// Mitsubishi GX Developer project: 中間搬送   PLC: Q02

PROGRAM MAIN
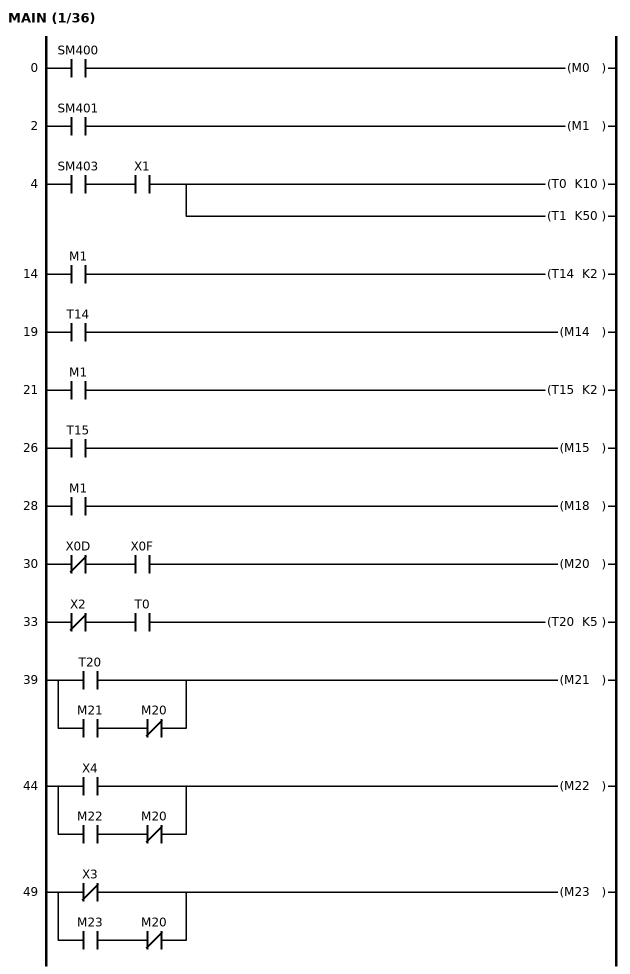
0     LD      SM400
      OUT     M0
2     LD      SM401
      OUT     M1
4     LD      SM403
      AND     X1
      OUT     T0 K10
      OUT     T1 K50
14    LD      M1
      OUT     T14 K2
19    LD      T14
      OUT     M14
21    LD      M1
      OUT     T15 K2
26    LD      T15
      OUT     M15
28    LD      M1
      OUT     M18
30    LDI     X0D
      AND     X0F
      OUT     M20
33    LDI     X2
      AND     T0
      OUT     T20 K5
39    LD      T20
      LD      M21
      ANI     M20
      ORB
      OUT     M21
44    LD      X4
      LD      M22
      ANI     M20
      ORB
      OUT     M22
49    LDI     X3
      LD      M23
      ANI     M20
      ORB
      OUT     M23
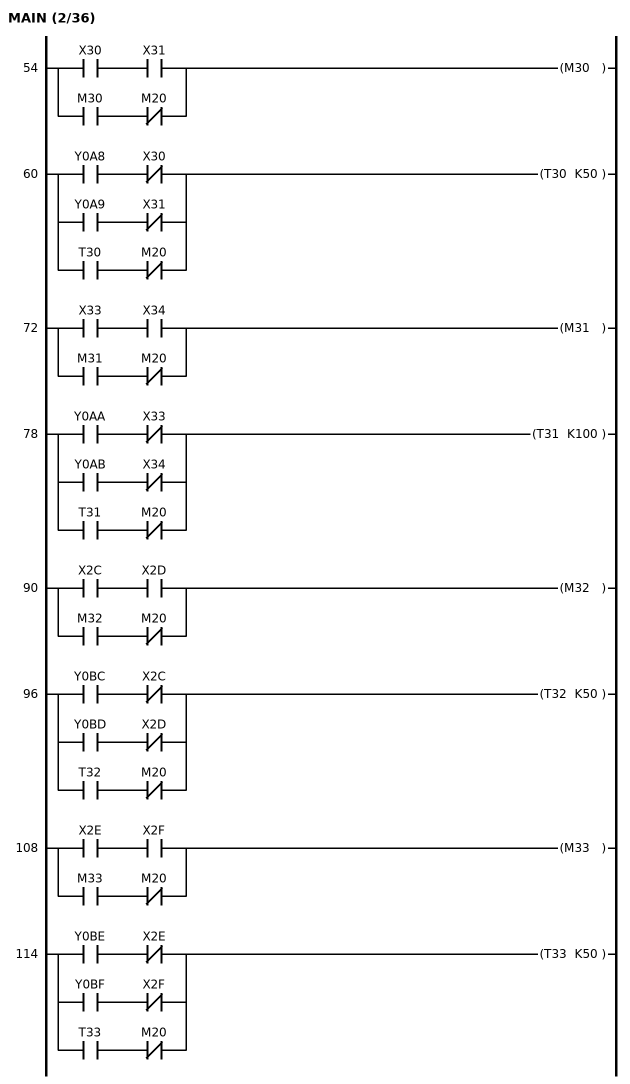
54    LD      X30
      AND     X31
      LD      M30
      ANI     M20
      ORB
      OUT     M30
60    LD      Y0A8
      ANI     X30
      LD      Y0A9
      ANI     X31
      ORB
      LD      T30
      ANI     M20
      ORB
      OUT     T30 K50
72    LD      X33
      AND     X34
      LD      M31
      ANI     M20
      ORB
      OUT     M31
78    LD      Y0AA
      ANI     X33
      LD      Y0AB
      ANI     X34
      ORB
      LD      T31
      ANI     M20
      ORB
      OUT     T31 K100
90    LD      X2C
      AND     X2D
      LD      M32
      ANI     M20
      ORB
      OUT     M32
96    LD      Y0BC
      ANI     X2C
      LD      Y0BD
      ANI     X2D
      ORB
      LD      T32
      ANI     M20
      ORB
      OUT     T32 K50
108   LD      X2E
      AND     X2F
      LD      M33
      ANI     M20
      ORB
      OUT     M33
114   LD      Y0BE
      ANI     X2E
      LD      Y0BF
      ANI     X2F
      ORB
      LD      T33
      ANI     M20
      ORB
      OUT     T33 K50
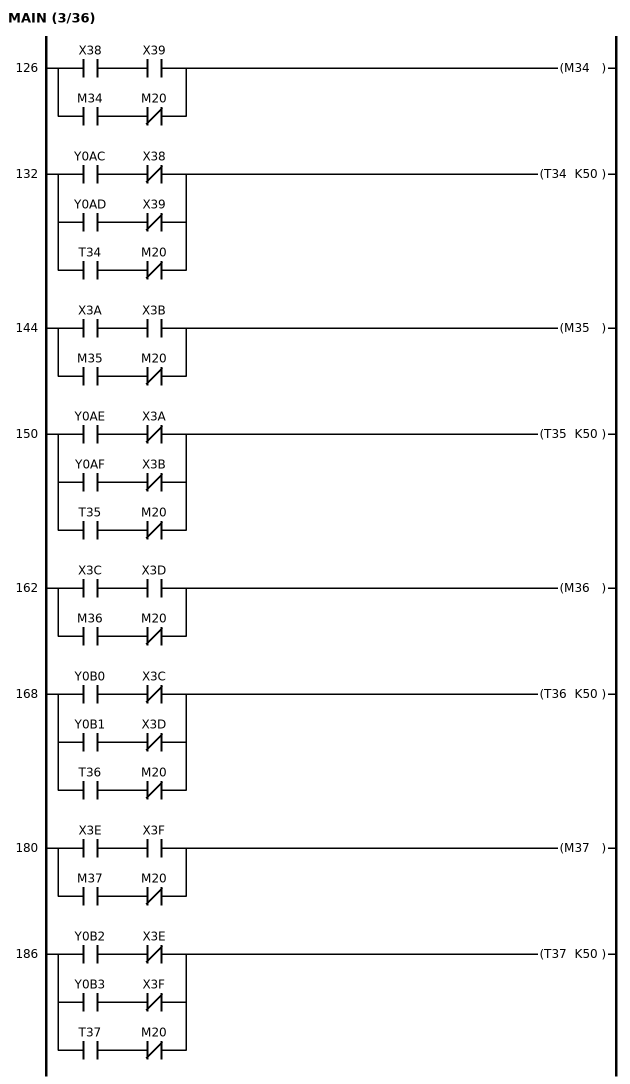
126   LD      X38
      AND     X39
      LD      M34
      ANI     M20
      ORB
      OUT     M34
132   LD      Y0AC
      ANI     X38
      LD      Y0AD
      ANI     X39
      ORB
      LD      T34
      ANI     M20
      ORB
      OUT     T34 K50
144   LD      X3A
      AND     X3B
      LD      M35
      ANI     M20
      ORB
      OUT     M35
150   LD      Y0AE
      ANI     X3A
      LD      Y0AF
      ANI     X3B
      ORB
      LD      T35
      ANI     M20
      ORB
      OUT     T35 K50
162   LD      X3C
      AND     X3D
      LD      M36
      ANI     M20
      ORB
      OUT     M36
168   LD      Y0B0
      ANI     X3C
      LD      Y0B1
      ANI     X3D
      ORB
      LD      T36
      ANI     M20
      ORB
      OUT     T36 K50
180   LD      X3E
      AND     X3F
      LD      M37
      ANI     M20
      ORB
      OUT     M37
186   LD      Y0B2
      ANI     X3E
      LD      Y0B3
      ANI     X3F
      ORB
      LD      T37
      ANI     M20
      ORB
      OUT     T37 K50
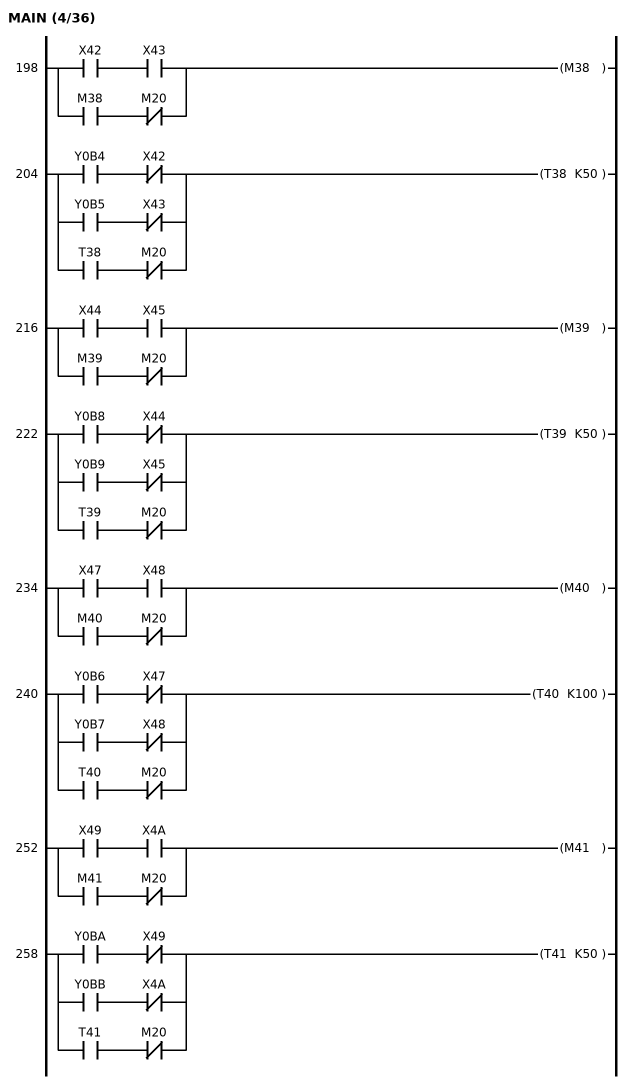
198   LD      X42
      AND     X43
      LD      M38
      ANI     M20
      ORB
      OUT     M38
204   LD      Y0B4
      ANI     X42
      LD      Y0B5
      ANI     X43
      ORB
      LD      T38
      ANI     M20
      ORB
      OUT     T38 K50
216   LD      X44
      AND     X45
      LD      M39
      ANI     M20
      ORB
      OUT     M39
222   LD      Y0B8
      ANI     X44
      LD      Y0B9
      ANI     X45
      ORB
      LD      T39
      ANI     M20
      ORB
      OUT     T39 K50
234   LD      X47
      AND     X48
      LD      M40
      ANI     M20
      ORB
      OUT     M40
240   LD      Y0B6
      ANI     X47
      LD      Y0B7
      ANI     X48
      ORB
      LD      T40
      ANI     M20
      ORB
      OUT     T40 K100
252   LD      X49
      AND     X4A
      LD      M41
      ANI     M20
      ORB
      OUT     M41
258   LD      Y0BA
      ANI     X49
      LD      Y0BB
      ANI     X4A
      ORB
      LD      T41
      ANI     M20
      ORB
      OUT     T41 K50
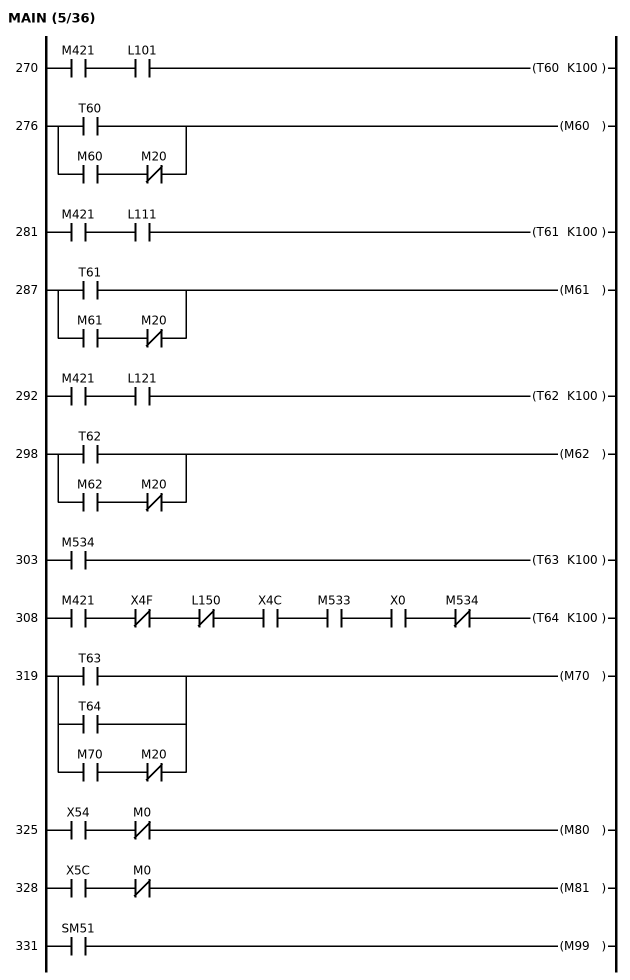
270   LD      M421
      AND     L101
      OUT     T60 K100
276   LD      T60
      LD      M60
      ANI     M20
      ORB
      OUT     M60
281   LD      M421
      AND     L111
      OUT     T61 K100
287   LD      T61
      LD      M61
      ANI     M20
      ORB
      OUT     M61
292   LD      M421
      AND     L121
      OUT     T62 K100
298   LD      T62
      LD      M62
      ANI     M20
      ORB
      OUT     M62
303   LD      M534
      OUT     T63 K100
308   LD      M421
      ANI     X4F
      ANI     L150
      AND     X4C
      AND     M533
      AND     X0
      ANI     M534
      OUT     T64 K100
319   LD      T63
      OR      T64
      LD      M70
      ANI     M20
      ORB
      OUT     M70
325   LD      X54
      ANI     M0
      OUT     M80
328   LD      X5C
      ANI     M0
      OUT     M81
331   LD      SM51
      OUT     M99
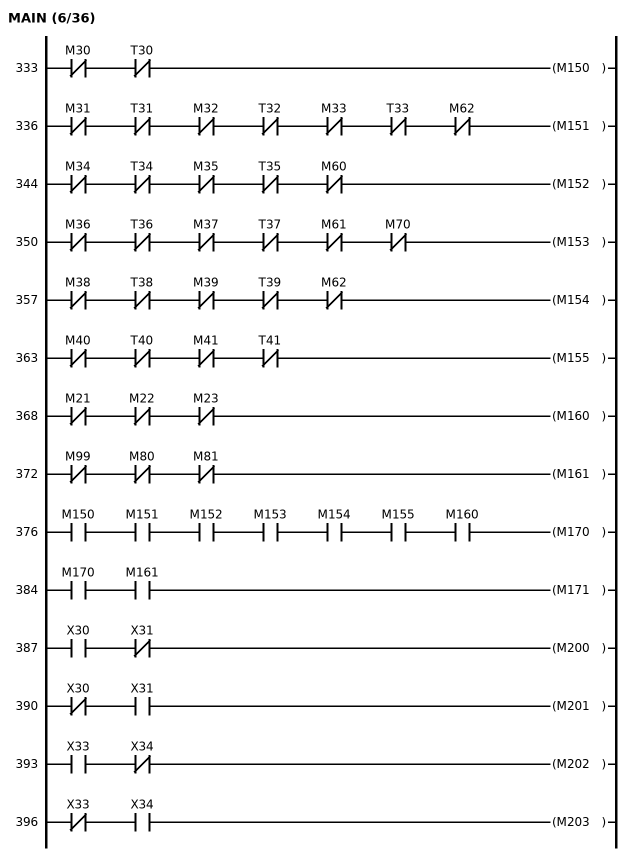
333   LDI     M30
      ANI     T30
      OUT     M150
336   LDI     M31
      ANI     T31
      ANI     M32
      ANI     T32
      ANI     M33
      ANI     T33
      ANI     M62
      OUT     M151
344   LDI     M34
      ANI     T34
      ANI     M35
      ANI     T35
      ANI     M60
      OUT     M152
350   LDI     M36
      ANI     T36
      ANI     M37
      ANI     T37
      ANI     M61
      ANI     M70
      OUT     M153
357   LDI     M38
      ANI     T38
      ANI     M39
      ANI     T39
      ANI     M62
      OUT     M154
363   LDI     M40
      ANI     T40
      ANI     M41
      ANI     T41
      OUT     M155
368   LDI     M21
      ANI     M22
      ANI     M23
      OUT     M160
372   LDI     M99
      ANI     M80
      ANI     M81
      OUT     M161
376   LD      M150
      AND     M151
      AND     M152
      AND     M153
      AND     M154
      AND     M155
      AND     M160
      OUT     M170
384   LD      M170
      AND     M161
      OUT     M171
387   LD      X30
      ANI     X31
      OUT     M200
390   LDI     X30
      AND     X31
      OUT     M201
393   LD      X33
      ANI     X34
      OUT     M202
396   LDI     X33
      AND     X34
      OUT     M203
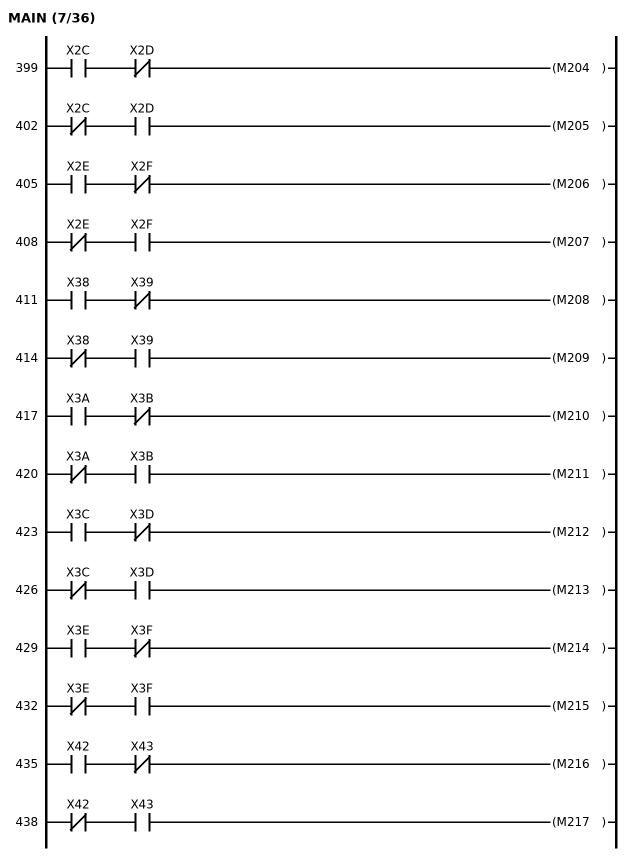
399   LD      X2C
      ANI     X2D
      OUT     M204
402   LDI     X2C
      AND     X2D
      OUT     M205
405   LD      X2E
      ANI     X2F
      OUT     M206
408   LDI     X2E
      AND     X2F
      OUT     M207
411   LD      X38
      ANI     X39
      OUT     M208
414   LDI     X38
      AND     X39
      OUT     M209
417   LD      X3A
      ANI     X3B
      OUT     M210
420   LDI     X3A
      AND     X3B
      OUT     M211
423   LD      X3C
      ANI     X3D
      OUT     M212
426   LDI     X3C
      AND     X3D
      OUT     M213
429   LD      X3E
      ANI     X3F
      OUT     M214
432   LDI     X3E
      AND     X3F
      OUT     M215
435   LD      X42
      ANI     X43
      OUT     M216
438   LDI     X42
      AND     X43
      OUT     M217
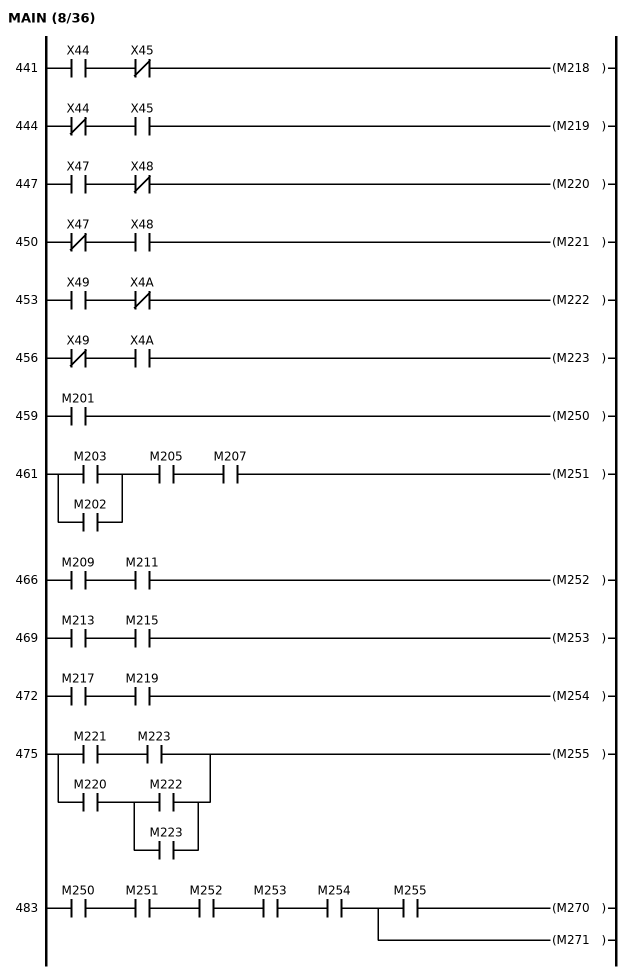
441   LD      X44
      ANI     X45
      OUT     M218
444   LDI     X44
      AND     X45
      OUT     M219
447   LD      X47
      ANI     X48
      OUT     M220
450   LDI     X47
      AND     X48
      OUT     M221
453   LD      X49
      ANI     X4A
      OUT     M222
456   LDI     X49
      AND     X4A
      OUT     M223
459   LD      M201
      OUT     M250
461   LD      M203
      OR      M202
      AND     M205
      AND     M207
      OUT     M251
466   LD      M209
      AND     M211
      OUT     M252
469   LD      M213
      AND     M215
      OUT     M253
472   LD      M217
      AND     M219
      OUT     M254
475   LD      M221
      AND     M223
      LD      M220
      LD      M222
      OR      M223
      ANB
      ORB
      OUT     M255
483   LD      M250
      AND     M251
      AND     M252
      AND     M253
      AND     M254
      MPS
      AND     M255
      OUT     M270
      MPP
      OUT     M271
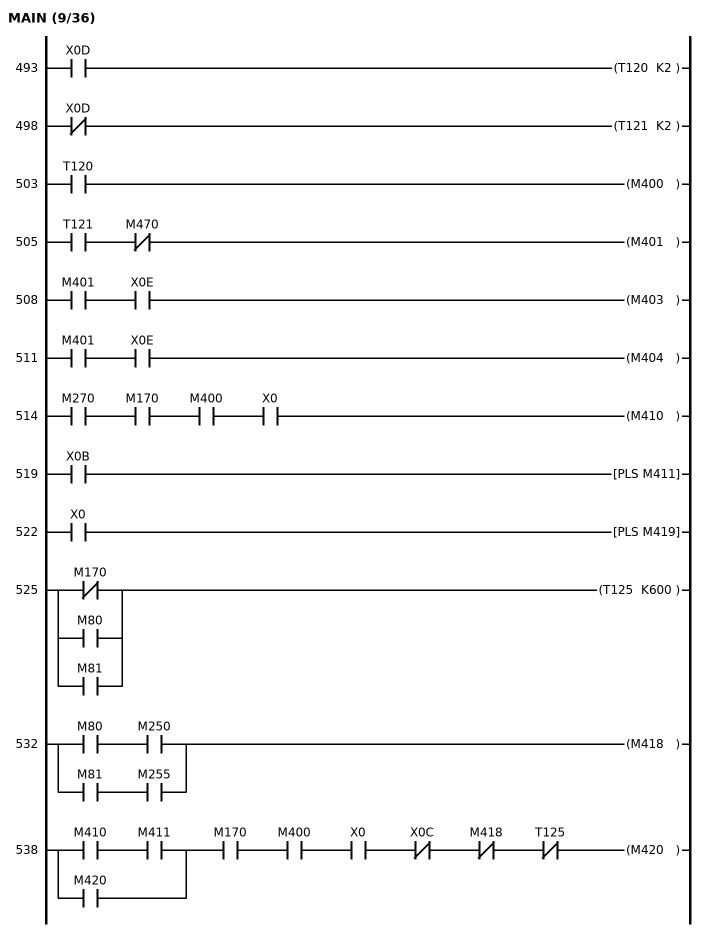
493   LD      X0D
      OUT     T120 K2
498   LDI     X0D
      OUT     T121 K2
503   LD      T120
      OUT     M400
505   LD      T121
      ANI     M470
      OUT     M401
508   LD      M401
      AND     X0E
      OUT     M403
511   LD      M401
      AND     X0E
      OUT     M404
514   LD      M270
      AND     M170
      AND     M400
      AND     X0
      OUT     M410
519   LD      X0B
      PLS     M411
522   LD      X0
      PLS     M419
525   LDI     M170
      OR      M80
      OR      M81
      OUT     T125 K600
532   LD      M80
      AND     M250
      LD      M81
      AND     M255
      ORB
      OUT     M418
538   LD      M410
      AND     M411
      OR      M420
      AND     M170
      AND     M400
      AND     X0
      ANI     X0C
      ANI     M418
      ANI     T125
      OUT     M420
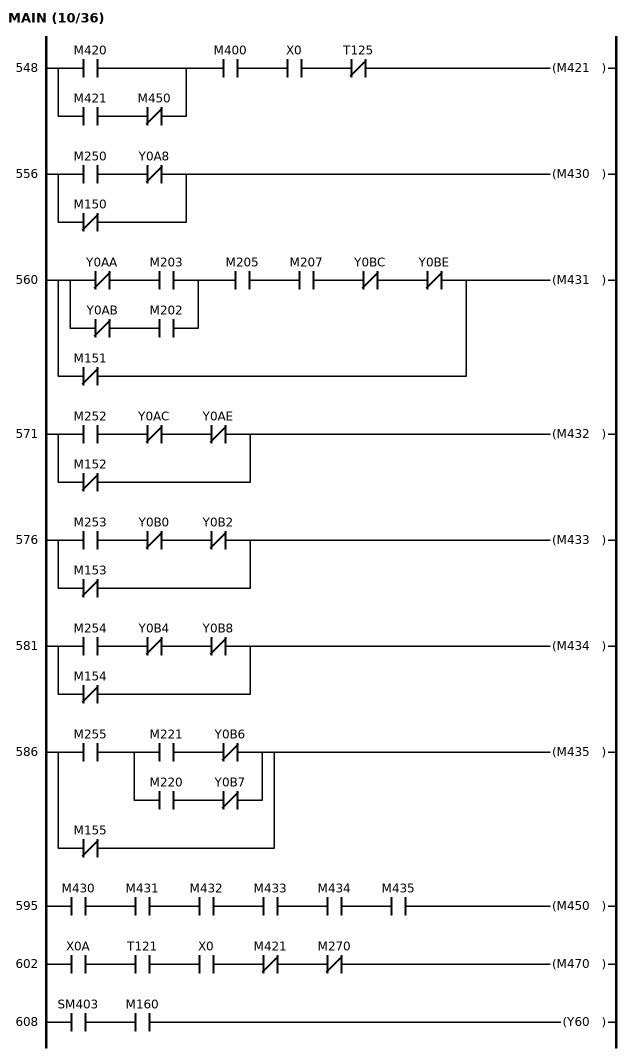
548   LD      M420
      LD      M421
      ANI     M450
      ORB
      AND     M400
      AND     X0
      ANI     T125
      OUT     M421
556   LD      M250
      ANI     Y0A8
      ORI     M150
      OUT     M430
560   LDI     Y0AA
      AND     M203
      LDI     Y0AB
      AND     M202
      ORB
      AND     M205
      AND     M207
      ANI     Y0BC
      ANI     Y0BE
      ORI     M151
      OUT     M431
571   LD      M252
      ANI     Y0AC
      ANI     Y0AE
      ORI     M152
      OUT     M432
576   LD      M253
      ANI     Y0B0
      ANI     Y0B2
      ORI     M153
      OUT     M433
581   LD      M254
      ANI     Y0B4
      ANI     Y0B8
      ORI     M154
      OUT     M434
586   LD      M255
      LD      M221
      ANI     Y0B6
      LD      M220
      ANI     Y0B7
      ORB
      ANB
      ORI     M155
      OUT     M435
595   LD      M430
      AND     M431
      AND     M432
      AND     M433
      AND     M434
      AND     M435
      OUT     M450
602   LD      X0A
      AND     T121
      AND     X0
      ANI     M421
      ANI     M270
      OUT     M470
608   LD      SM403
      AND     M160
      OUT     Y60
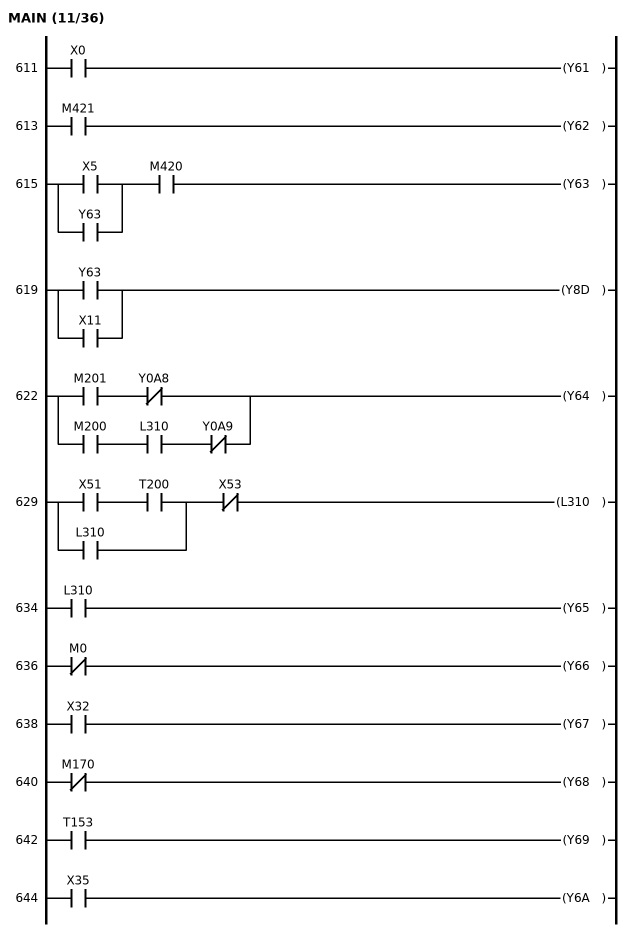
611   LD      X0
      OUT     Y61
613   LD      M421
      OUT     Y62
615   LD      X5
      OR      Y63
      AND     M420
      OUT     Y63
619   LD      Y63
      OR      X11
      OUT     Y8D
622   LD      M201
      ANI     Y0A8
      LD      M200
      AND     L310
      ANI     Y0A9
      ORB
      OUT     Y64
629   LD      X51
      AND     T200
      OR      L310
      ANI     X53
      OUT     L310
634   LD      L310
      OUT     Y65
636   LDI     M0
      OUT     Y66
638   LD      X32
      OUT     Y67
640   LDI     M170
      OUT     Y68
642   LD      T153
      OUT     Y69
644   LD      X35
      OUT     Y6A
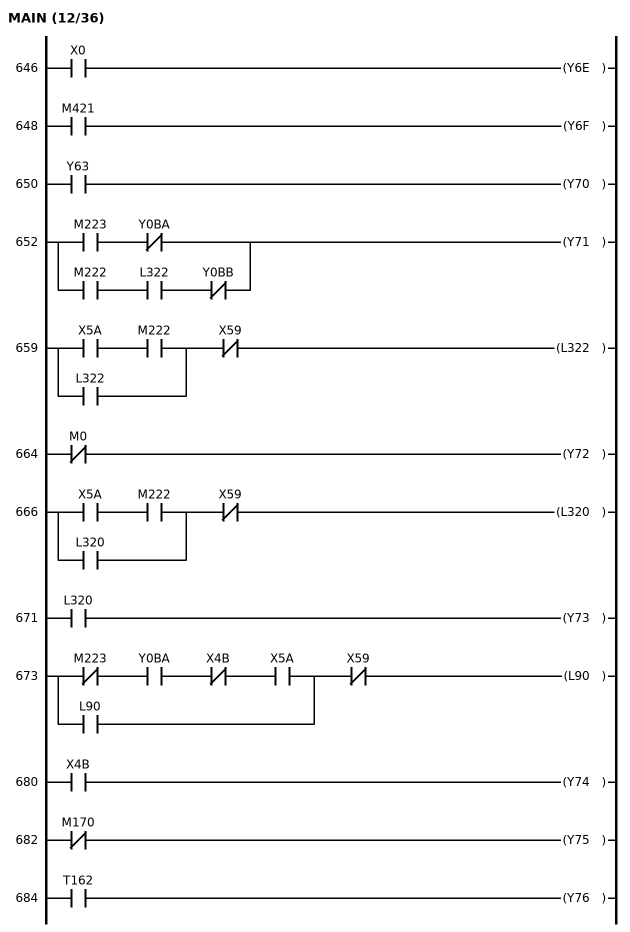
646   LD      X0
      OUT     Y6E
648   LD      M421
      OUT     Y6F
650   LD      Y63
      OUT     Y70
652   LD      M223
      ANI     Y0BA
      LD      M222
      AND     L322
      ANI     Y0BB
      ORB
      OUT     Y71
659   LD      X5A
      AND     M222
      OR      L322
      ANI     X59
      OUT     L322
664   LDI     M0
      OUT     Y72
666   LD      X5A
      AND     M222
      OR      L320
      ANI     X59
      OUT     L320
671   LD      L320
      OUT     Y73
673   LDI     M223
      AND     Y0BA
      ANI     X4B
      AND     X5A
      OR      L90
      ANI     X59
      OUT     L90
680   LD      X4B
      OUT     Y74
682   LDI     M170
      OUT     Y75
684   LD      T162
      OUT     Y76
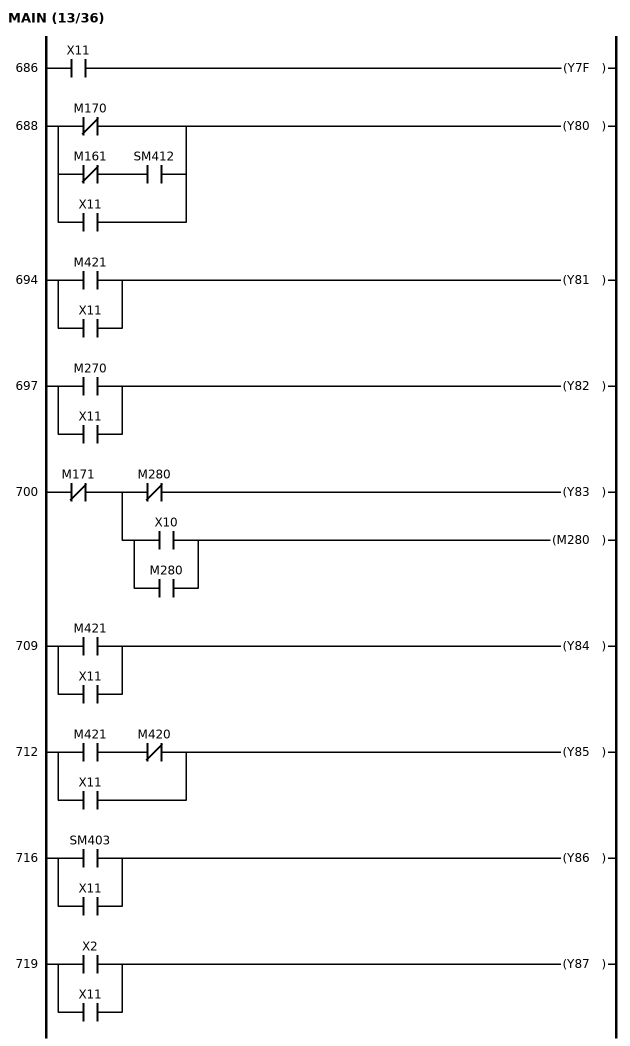
686   LD      X11
      OUT     Y7F
688   LDI     M170
      LDI     M161
      AND     SM412
      ORB
      OR      X11
      OUT     Y80
694   LD      M421
      OR      X11
      OUT     Y81
697   LD      M270
      OR      X11
      OUT     Y82
700   LDI     M171
      MPS
      ANI     M280
      OUT     Y83
      MPP
      LD      X10
      OR      M280
      ANB
      OUT     M280
709   LD      M421
      OR      X11
      OUT     Y84
712   LD      M421
      ANI     M420
      OR      X11
      OUT     Y85
716   LD      SM403
      OR      X11
      OUT     Y86
719   LD      X2
      OR      X11
      OUT     Y87
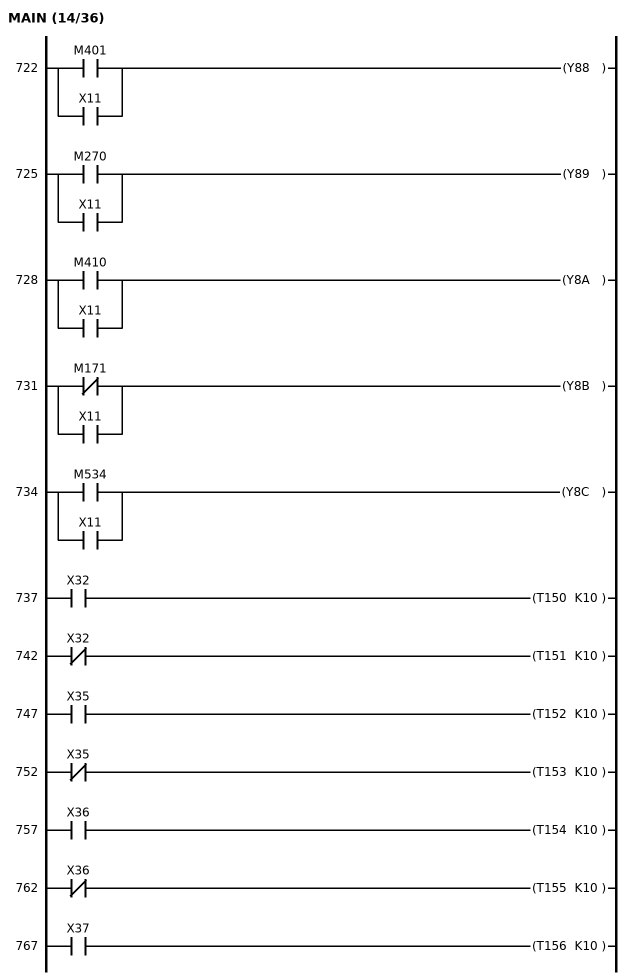
722   LD      M401
      OR      X11
      OUT     Y88
725   LD      M270
      OR      X11
      OUT     Y89
728   LD      M410
      OR      X11
      OUT     Y8A
731   LDI     M171
      OR      X11
      OUT     Y8B
734   LD      M534
      OR      X11
      OUT     Y8C
737   LD      X32
      OUT     T150 K10
742   LDI     X32
      OUT     T151 K10
747   LD      X35
      OUT     T152 K10
752   LDI     X35
      OUT     T153 K10
757   LD      X36
      OUT     T154 K10
762   LDI     X36
      OUT     T155 K10
767   LD      X37
      OUT     T156 K10
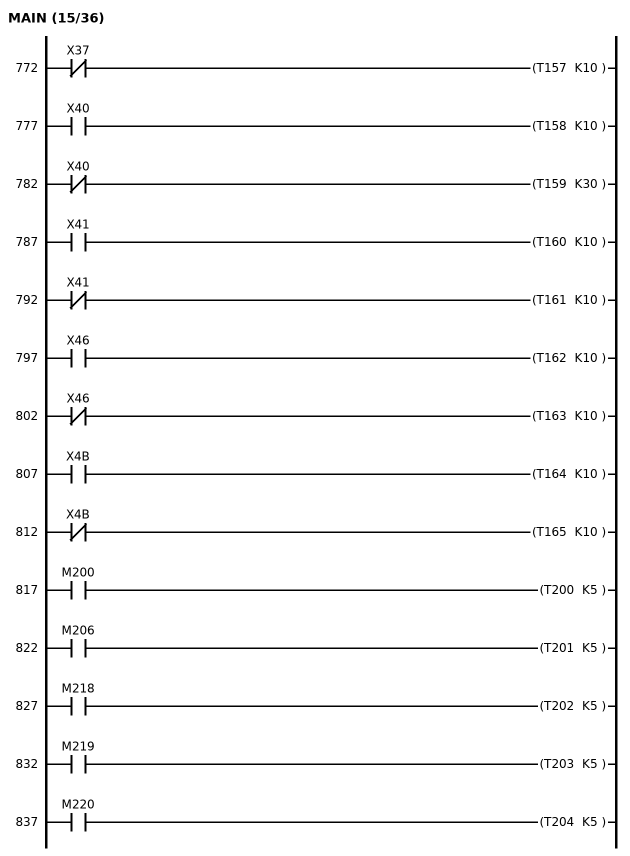
772   LDI     X37
      OUT     T157 K10
777   LD      X40
      OUT     T158 K10
782   LDI     X40
      OUT     T159 K30
787   LD      X41
      OUT     T160 K10
792   LDI     X41
      OUT     T161 K10
797   LD      X46
      OUT     T162 K10
802   LDI     X46
      OUT     T163 K10
807   LD      X4B
      OUT     T164 K10
812   LDI     X4B
      OUT     T165 K10
817   LD      M200
      OUT     T200 K5
822   LD      M206
      OUT     T201 K5
827   LD      M218
      OUT     T202 K5
832   LD      M219
      OUT     T203 K5
837   LD      M220
      OUT     T204 K5
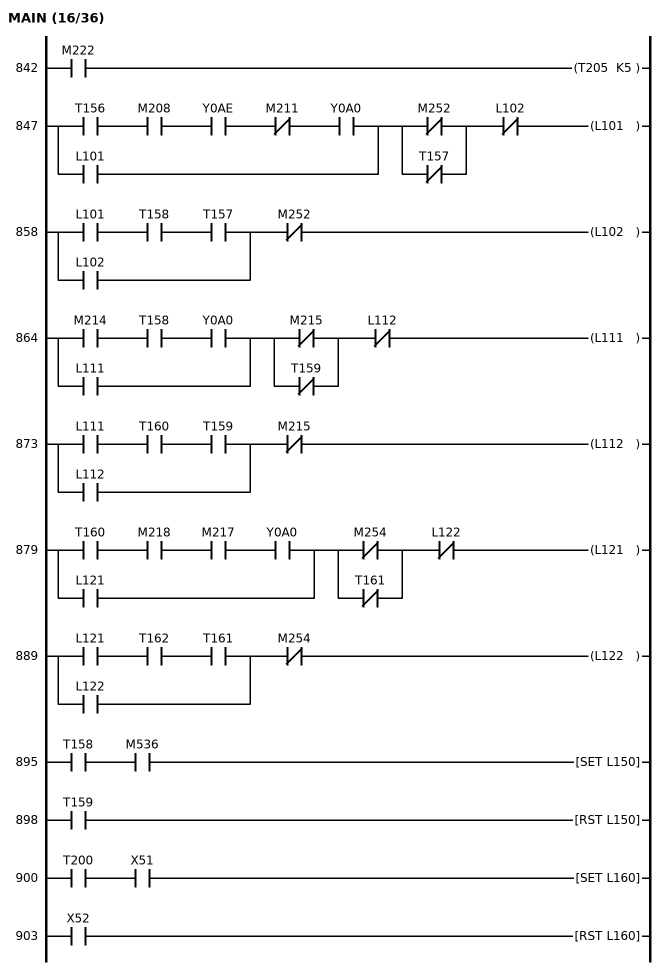
842   LD      M222
      OUT     T205 K5
847   LD      T156
      AND     M208
      AND     Y0AE
      ANI     M211
      AND     Y0A0
      OR      L101
      LDI     M252
      ORI     T157
      ANB
      ANI     L102
      OUT     L101
858   LD      L101
      AND     T158
      AND     T157
      OR      L102
      ANI     M252
      OUT     L102
864   LD      M214
      AND     T158
      AND     Y0A0
      OR      L111
      LDI     M215
      ORI     T159
      ANB
      ANI     L112
      OUT     L111
873   LD      L111
      AND     T160
      AND     T159
      OR      L112
      ANI     M215
      OUT     L112
879   LD      T160
      AND     M218
      AND     M217
      AND     Y0A0
      OR      L121
      LDI     M254
      ORI     T161
      ANB
      ANI     L122
      OUT     L121
889   LD      L121
      AND     T162
      AND     T161
      OR      L122
      ANI     M254
      OUT     L122
895   LD      T158
      AND     M536
      SET     L150
898   LD      T159
      RST     L150
900   LD      T200
      AND     X51
      SET     L160
903   LD      X52
      RST     L160
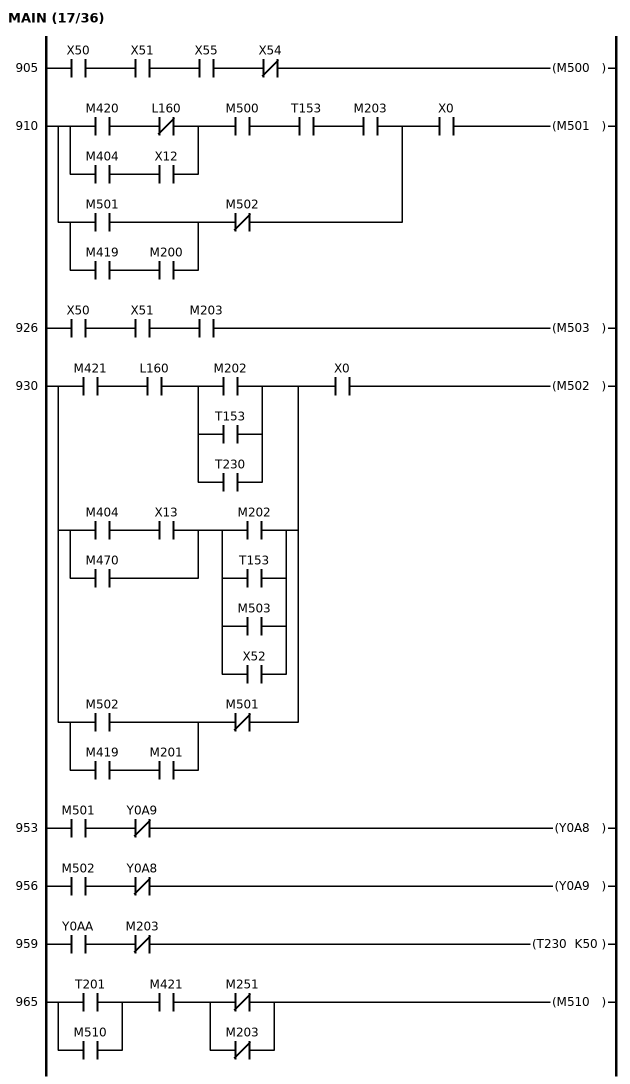
905   LD      X50
      AND     X51
      AND     X55
      ANI     X54
      OUT     M500
910   LD      M420
      ANI     L160
      LD      M404
      AND     X12
      ORB
      AND     M500
      AND     T153
      AND     M203
      LD      M501
      LD      M419
      AND     M200
      ORB
      ANI     M502
      ORB
      AND     X0
      OUT     M501
926   LD      X50
      AND     X51
      AND     M203
      OUT     M503
930   LD      M421
      AND     L160
      LD      M202
      OR      T153
      OR      T230
      ANB
      LD      M404
      AND     X13
      OR      M470
      LD      M202
      OR      T153
      OR      M503
      OR      X52
      ANB
      ORB
      LD      M502
      LD      M419
      AND     M201
      ORB
      ANI     M501
      ORB
      AND     X0
      OUT     M502
953   LD      M501
      ANI     Y0A9
      OUT     Y0A8
956   LD      M502
      ANI     Y0A8
      OUT     Y0A9
959   LD      Y0AA
      ANI     M203
      OUT     T230 K50
965   LD      T201
      OR      M510
      AND     M421
      LDI     M251
      ORI     M203
      ANB
      OUT     M510
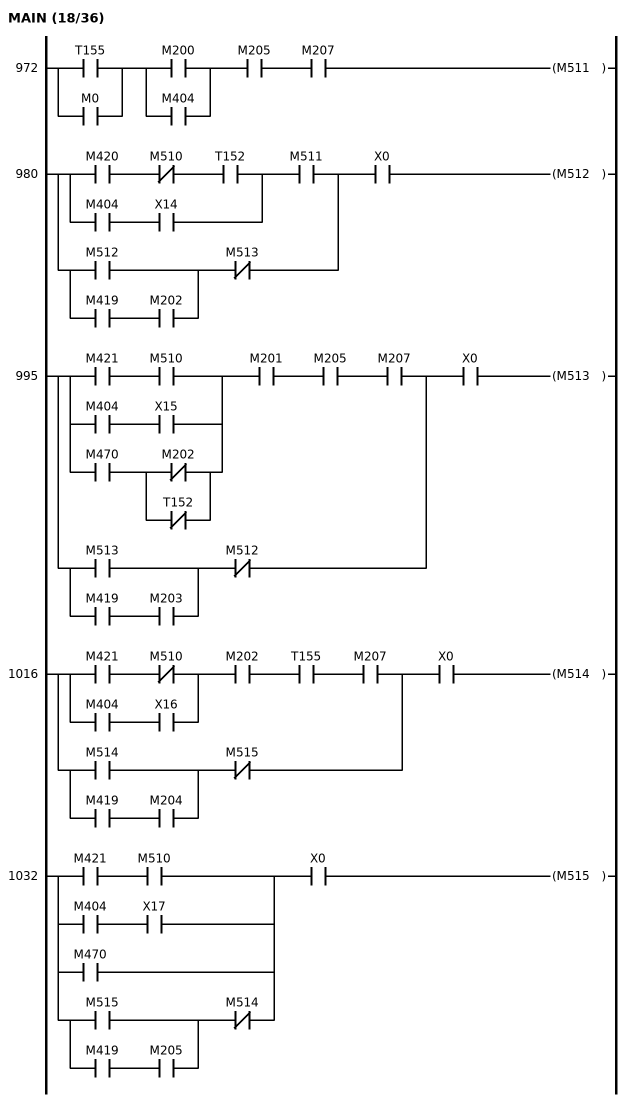
972   LD      T155
      OR      M0
      LD      M200
      OR      M404
      ANB
      AND     M205
      AND     M207
      OUT     M511
980   LD      M420
      ANI     M510
      AND     T152
      LD      M404
      AND     X14
      ORB
      AND     M511
      LD      M512
      LD      M419
      AND     M202
      ORB
      ANI     M513
      ORB
      AND     X0
      OUT     M512
995   LD      M421
      AND     M510
      LD      M404
      AND     X15
      ORB
      LD      M470
      LDI     M202
      ORI     T152
      ANB
      ORB
      AND     M201
      AND     M205
      AND     M207
      LD      M513
      LD      M419
      AND     M203
      ORB
      ANI     M512
      ORB
      AND     X0
      OUT     M513
1016  LD      M421
      ANI     M510
      LD      M404
      AND     X16
      ORB
      AND     M202
      AND     T155
      AND     M207
      LD      M514
      LD      M419
      AND     M204
      ORB
      ANI     M515
      ORB
      AND     X0
      OUT     M514
1032  LD      M421
      AND     M510
      LD      M404
      AND     X17
      ORB
      OR      M470
      LD      M515
      LD      M419
      AND     M205
      ORB
      ANI     M514
      ORB
      AND     X0
      OUT     M515
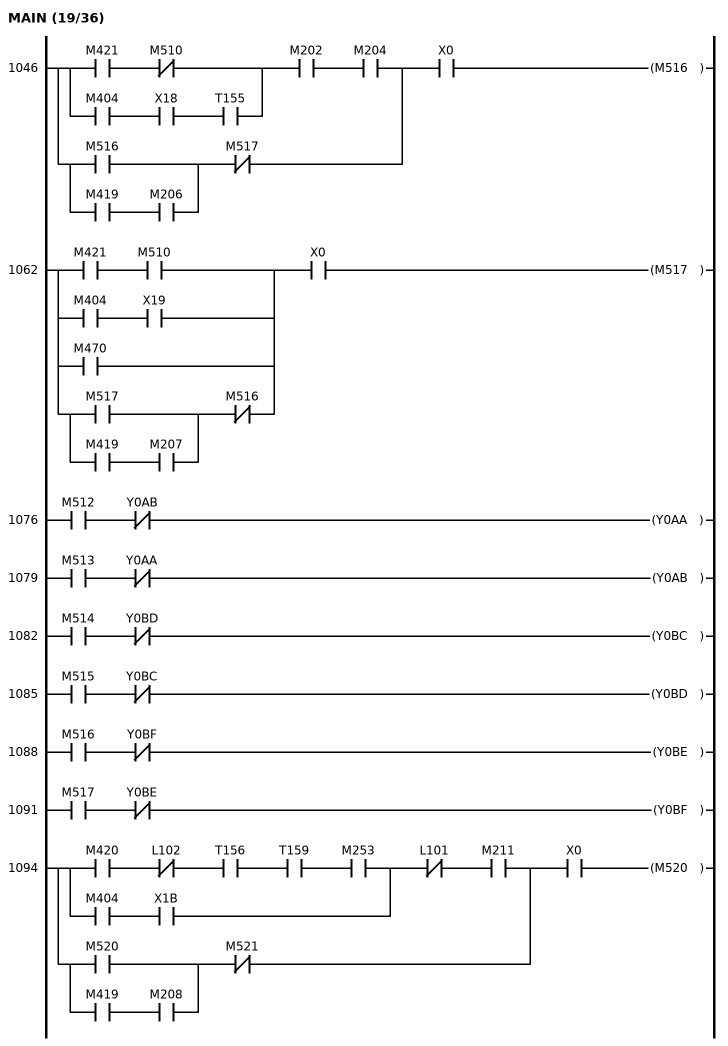
1046  LD      M421
      ANI     M510
      LD      M404
      AND     X18
      AND     T155
      ORB
      AND     M202
      AND     M204
      LD      M516
      LD      M419
      AND     M206
      ORB
      ANI     M517
      ORB
      AND     X0
      OUT     M516
1062  LD      M421
      AND     M510
      LD      M404
      AND     X19
      ORB
      OR      M470
      LD      M517
      LD      M419
      AND     M207
      ORB
      ANI     M516
      ORB
      AND     X0
      OUT     M517
1076  LD      M512
      ANI     Y0AB
      OUT     Y0AA
1079  LD      M513
      ANI     Y0AA
      OUT     Y0AB
1082  LD      M514
      ANI     Y0BD
      OUT     Y0BC
1085  LD      M515
      ANI     Y0BC
      OUT     Y0BD
1088  LD      M516
      ANI     Y0BF
      OUT     Y0BE
1091  LD      M517
      ANI     Y0BE
      OUT     Y0BF
1094  LD      M420
      ANI     L102
      AND     T156
      AND     T159
      AND     M253
      LD      M404
      AND     X1B
      ORB
      ANI     L101
      AND     M211
      LD      M520
      LD      M419
      AND     M208
      ORB
      ANI     M521
      ORB
      AND     X0
      OUT     M520
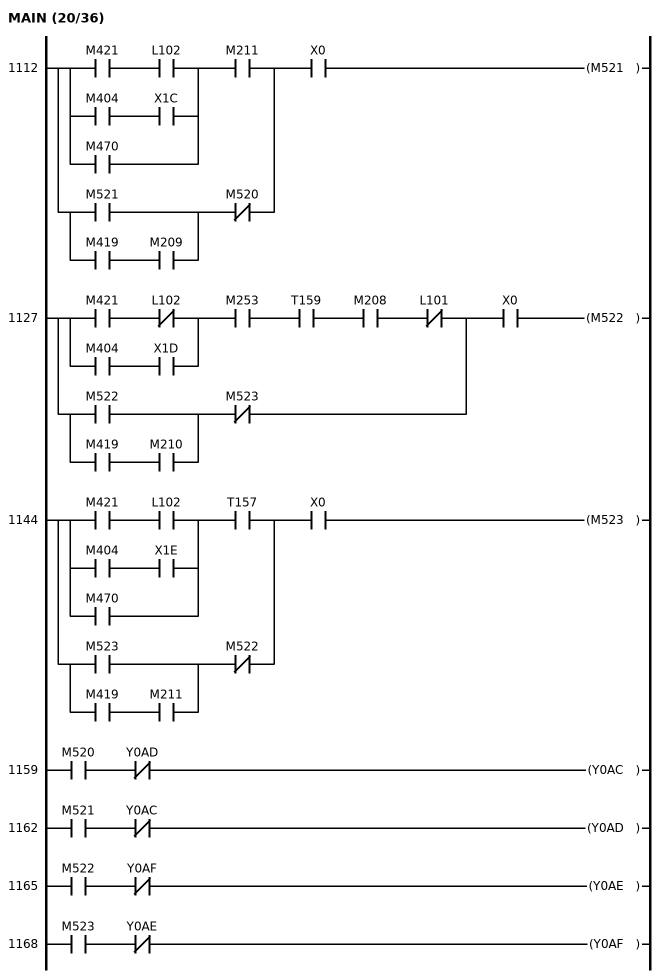
1112  LD      M421
      AND     L102
      LD      M404
      AND     X1C
      ORB
      OR      M470
      AND     M211
      LD      M521
      LD      M419
      AND     M209
      ORB
      ANI     M520
      ORB
      AND     X0
      OUT     M521
1127  LD      M421
      ANI     L102
      LD      M404
      AND     X1D
      ORB
      AND     M253
      AND     T159
      AND     M208
      ANI     L101
      LD      M522
      LD      M419
      AND     M210
      ORB
      ANI     M523
      ORB
      AND     X0
      OUT     M522
1144  LD      M421
      AND     L102
      LD      M404
      AND     X1E
      ORB
      OR      M470
      AND     T157
      LD      M523
      LD      M419
      AND     M211
      ORB
      ANI     M522
      ORB
      AND     X0
      OUT     M523
1159  LD      M520
      ANI     Y0AD
      OUT     Y0AC
1162  LD      M521
      ANI     Y0AC
      OUT     Y0AD
1165  LD      M522
      ANI     Y0AF
      OUT     Y0AE
1168  LD      M523
      ANI     Y0AE
      OUT     Y0AF
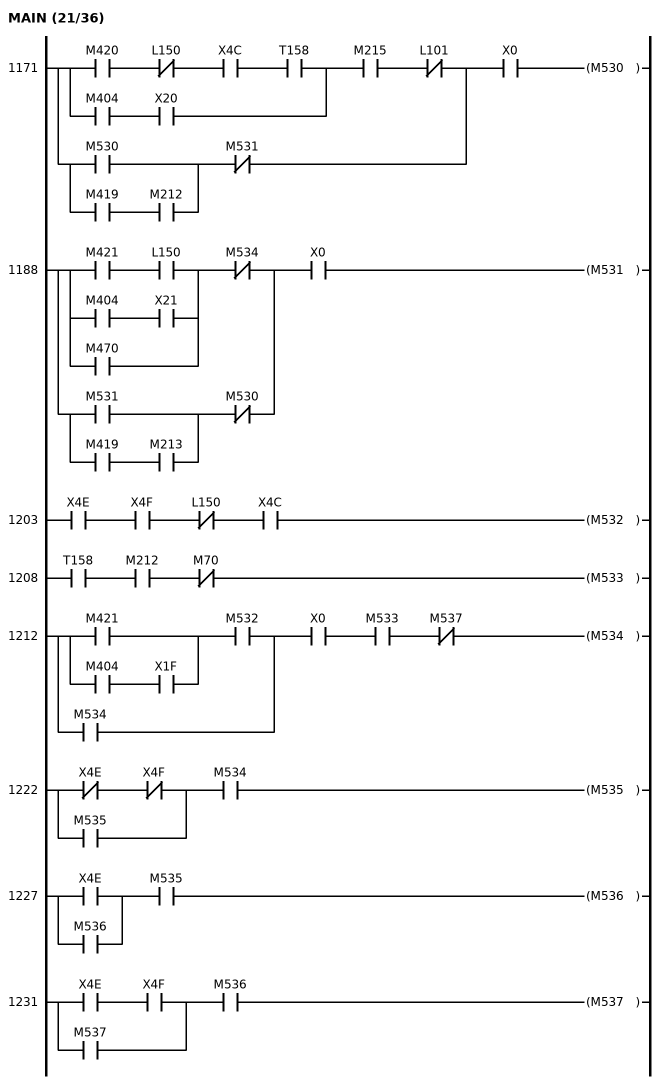
1171  LD      M420
      ANI     L150
      AND     X4C
      AND     T158
      LD      M404
      AND     X20
      ORB
      AND     M215
      ANI     L101
      LD      M530
      LD      M419
      AND     M212
      ORB
      ANI     M531
      ORB
      AND     X0
      OUT     M530
1188  LD      M421
      AND     L150
      LD      M404
      AND     X21
      ORB
      OR      M470
      ANI     M534
      LD      M531
      LD      M419
      AND     M213
      ORB
      ANI     M530
      ORB
      AND     X0
      OUT     M531
1203  LD      X4E
      AND     X4F
      ANI     L150
      AND     X4C
      OUT     M532
1208  LD      T158
      AND     M212
      ANI     M70
      OUT     M533
1212  LD      M421
      LD      M404
      AND     X1F
      ORB
      AND     M532
      OR      M534
      AND     X0
      AND     M533
      ANI     M537
      OUT     M534
1222  LDI     X4E
      ANI     X4F
      OR      M535
      AND     M534
      OUT     M535
1227  LD      X4E
      OR      M536
      AND     M535
      OUT     M536
1231  LD      X4E
      AND     X4F
      OR      M537
      AND     M536
      OUT     M537
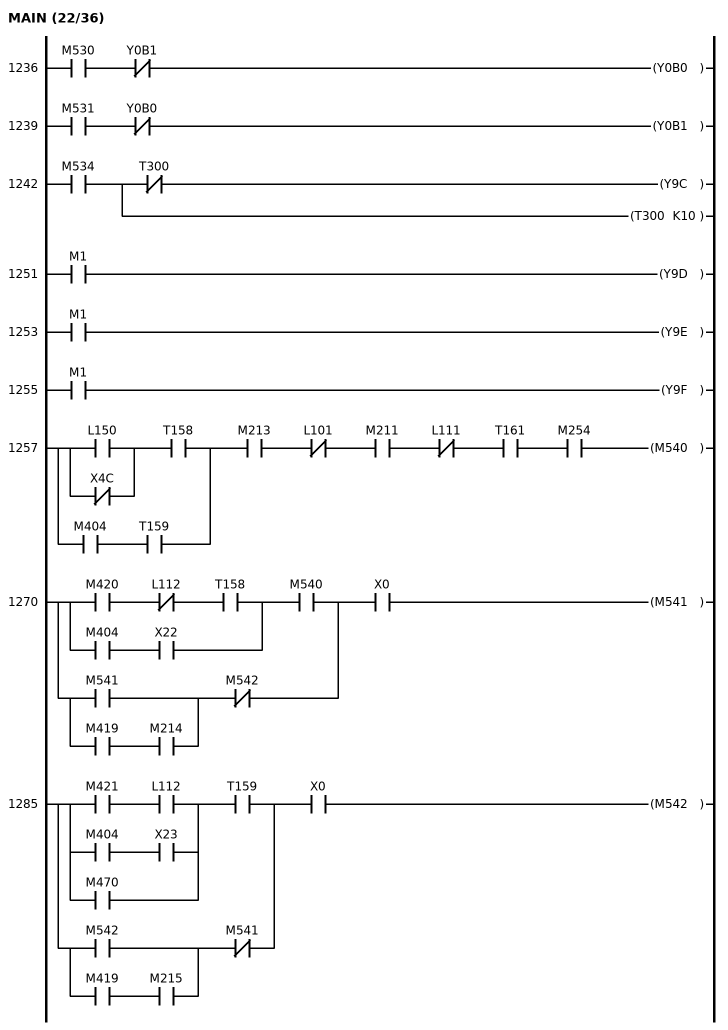
1236  LD      M530
      ANI     Y0B1
      OUT     Y0B0
1239  LD      M531
      ANI     Y0B0
      OUT     Y0B1
1242  LD      M534
      MPS
      ANI     T300
      OUT     Y9C
      MPP
      OUT     T300 K10
1251  LD      M1
      OUT     Y9D
1253  LD      M1
      OUT     Y9E
1255  LD      M1
      OUT     Y9F
1257  LD      L150
      ORI     X4C
      AND     T158
      LD      M404
      AND     T159
      ORB
      AND     M213
      ANI     L101
      AND     M211
      ANI     L111
      AND     T161
      AND     M254
      OUT     M540
1270  LD      M420
      ANI     L112
      AND     T158
      LD      M404
      AND     X22
      ORB
      AND     M540
      LD      M541
      LD      M419
      AND     M214
      ORB
      ANI     M542
      ORB
      AND     X0
      OUT     M541
1285  LD      M421
      AND     L112
      LD      M404
      AND     X23
      ORB
      OR      M470
      AND     T159
      LD      M542
      LD      M419
      AND     M215
      ORB
      ANI     M541
      ORB
      AND     X0
      OUT     M542
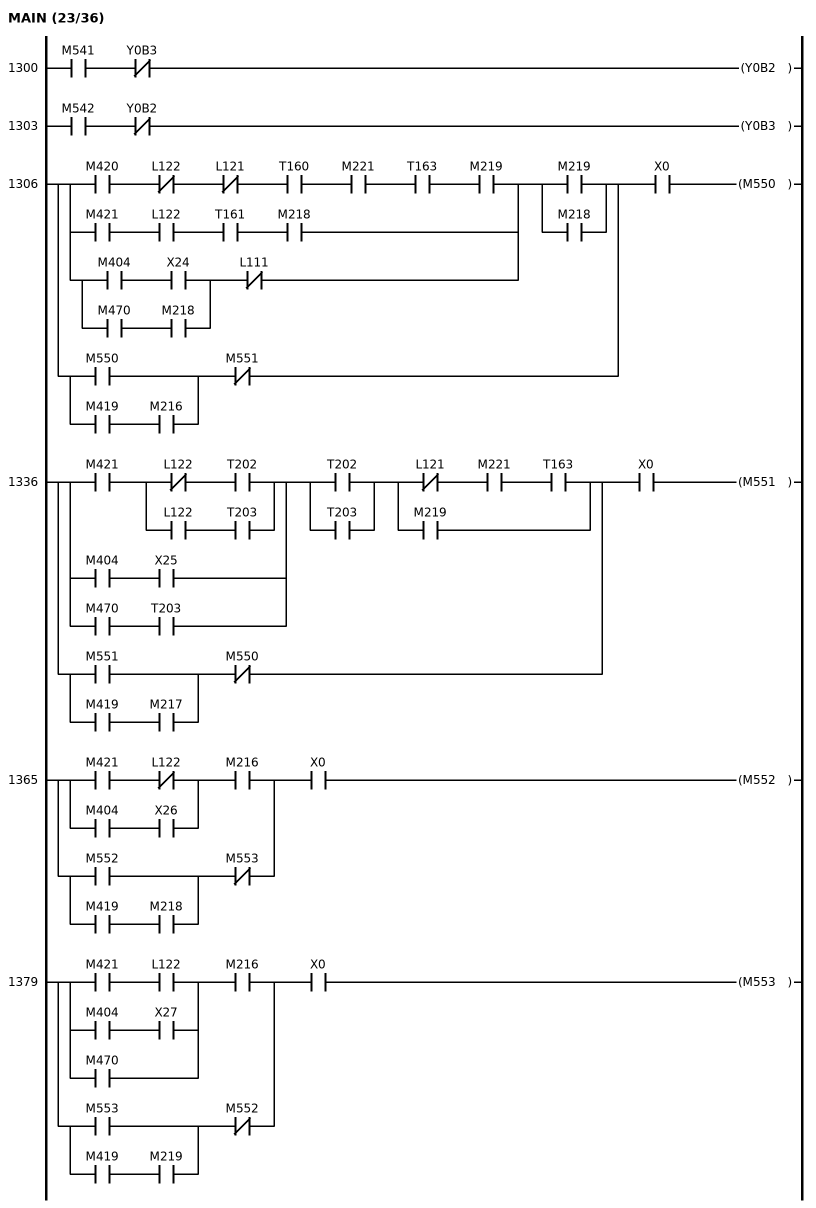
1300  LD      M541
      ANI     Y0B3
      OUT     Y0B2
1303  LD      M542
      ANI     Y0B2
      OUT     Y0B3
1306  LD      M420
      ANI     L122
      ANI     L121
      AND     T160
      AND     M221
      AND     T163
      AND     M219
      LD      M421
      AND     L122
      AND     T161
      AND     M218
      ORB
      LD      M404
      AND     X24
      LD      M470
      AND     M218
      ORB
      ANI     L111
      ORB
      LD      M219
      OR      M218
      ANB
      LD      M550
      LD      M419
      AND     M216
      ORB
      ANI     M551
      ORB
      AND     X0
      OUT     M550
1336  LD      M421
      LDI     L122
      AND     T202
      LD      L122
      AND     T203
      ORB
      ANB
      LD      M404
      AND     X25
      ORB
      LD      M470
      AND     T203
      ORB
      LD      T202
      OR      T203
      ANB
      LDI     L121
      AND     M221
      AND     T163
      OR      M219
      ANB
      LD      M551
      LD      M419
      AND     M217
      ORB
      ANI     M550
      ORB
      AND     X0
      OUT     M551
1365  LD      M421
      ANI     L122
      LD      M404
      AND     X26
      ORB
      AND     M216
      LD      M552
      LD      M419
      AND     M218
      ORB
      ANI     M553
      ORB
      AND     X0
      OUT     M552
1379  LD      M421
      AND     L122
      LD      M404
      AND     X27
      ORB
      OR      M470
      AND     M216
      LD      M553
      LD      M419
      AND     M219
      ORB
      ANI     M552
      ORB
      AND     X0
      OUT     M553
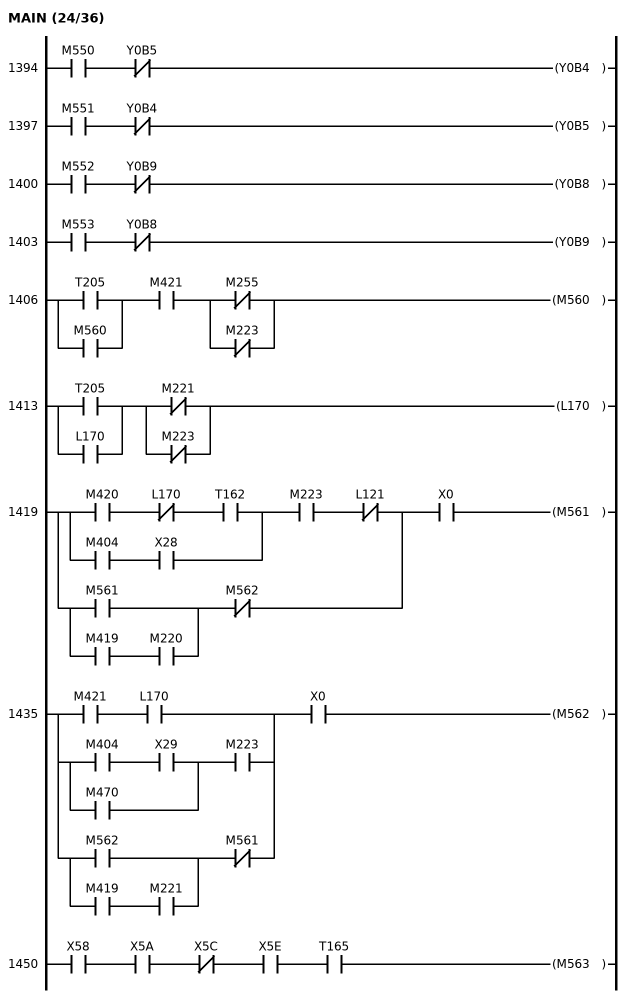
1394  LD      M550
      ANI     Y0B5
      OUT     Y0B4
1397  LD      M551
      ANI     Y0B4
      OUT     Y0B5
1400  LD      M552
      ANI     Y0B9
      OUT     Y0B8
1403  LD      M553
      ANI     Y0B8
      OUT     Y0B9
1406  LD      T205
      OR      M560
      AND     M421
      LDI     M255
      ORI     M223
      ANB
      OUT     M560
1413  LD      T205
      OR      L170
      LDI     M221
      ORI     M223
      ANB
      OUT     L170
1419  LD      M420
      ANI     L170
      AND     T162
      LD      M404
      AND     X28
      ORB
      AND     M223
      ANI     L121
      LD      M561
      LD      M419
      AND     M220
      ORB
      ANI     M562
      ORB
      AND     X0
      OUT     M561
1435  LD      M421
      AND     L170
      LD      M404
      AND     X29
      OR      M470
      AND     M223
      ORB
      LD      M562
      LD      M419
      AND     M221
      ORB
      ANI     M561
      ORB
      AND     X0
      OUT     M562
1450  LD      X58
      AND     X5A
      ANI     X5C
      AND     X5E
      AND     T165
      OUT     M563
